TYPE ST_HMI_CONTROL_SETTING_ITEM_OUT :
STRUCT
	stButtonSave		: ST_HMI_BUTTON_OUT;
	bVisible_RecipeMode	: BOOL;
	nRecipeMode			: INT; //count of recipe mode list
	aRecipeMode			: ARRAY[0..E_RecipeMode.eRecipeMode_Max] OF ST_Text;
	
	bVisible_UserLevel	: BOOL;
	bVisible_Bool		: BOOL;
	bVisible_Float		: BOOL;
	bVisible_Number		: BOOL;
	bVisible_String		: BOOL;
	bVisibleInfo		: BOOL;
	stInfo				: ST_Text;
	
	nUserLevelUsers		: INT; //count of recipe mode list
	aUserLevelUsers		: ARRAY[0..E_User_Level.eUser_Level_nMaxIdx] OF ST_Text;
END_STRUCT
END_TYPE

(* stored: Version 1.1.0.1, ProductVersion 3.1.4024.12
   DUT ST_HMI_CONTROL_SETTING_ITEM_OUT: Id {c6cd3180-2579-4600-86af-6f919aa18f78} *)
